(* IEC 61131-3 sources: Mizera_Tube/Plc (part 12) *)

(* ---- mac_func.plc ---- *)
*******************************************************************************
*   MAC_FUNC.PLC
*   ESAutomotion
*   LASER machine
*******************************************************************************
VAR
#include "cnc.inc"
END_VAR

VAR_IN_OUT
#include "mem.inc"
#include "RemContr.inc"
END_VAR

#include "iol.inc"

*******************************************************************************
* function block to manage the override
*******************************************************************************
FUNCTION_BLOCK OVERRIDE

VAR_INPUT
xAnalInput:          DWORD;     * input for potentiometer
xForceLowFeed:       BOOL;      * force the feed to SlowFeed
END_VAR

VAR_OUTPUT
y_Value:             DWORD;
END_VAR

VAR
feedVal:             DWORD;
TON_guiJOG_Min:        TON;   *TON for GUI button JOG to Minus
TON_guiJOG_Max:        TON;   *TON for GUI button JOG to Maximum
TON_BlinkAux_A:	       TON;   *TON Blinking Auxiliar Step A
TON_BlinkAux_B:	       TON;   *TON Blinking Auxiliar Step B
RTRG_guiJOG_Min:    R_TRIG;   *RTRIG for GUI button JOG to Minus
RTRG_guiJOG_Max:    R_TRIG;   *RTRIG for GUI button JOG to Maximum
RTRG_auxBlinkAux:   R_TRIG;
ValOvrr:             DWORD;   *DWORD Calculated value for Override from EncAPos
auxBlinkAux_A:        BOOL;   *BOOL Auxiliar Blinking 150 mseg Step A
auxBlinkAux_B:        BOOL;   *BOOL Auxiliar Blinking 150 mseg Step B
FeedGuiMem:          DWORD;   * support memory for hmi feedrate management
FEED_Minus:           BOOL;
FEED_Plus:            BOOL;

END_VAR
*******************************************************************************

LD   %Type
EQ   0
JMPCN no_analogue_sig

LD   xAnalInput                    ** input for potentiometer
MUL  %MaxPercent
DIV  4095                 *  (16 bit = 32767) [ se 12 bit usare 4095 ]
ST   feedVal              * DWORD Calculated value for Override

JMP  end
no_analogue_sig:

*-----------------------------------------------------------------
* FEED Override by GUI pushbuttons

LD   %Type
EQ   1
JMPCN no_HMI_sig

LD   %PulMinus             ** RTRIG for GUI button JOG to Minus
OR   RemContrFeedMinus     ** Xhc_Puls.13 Feed minus
ST   FEED_Minus

LD   %PulPlus              ** RTRIG for GUI button JOG to Maximum
OR   RemContrFeedPlus      ** Xhc_Puls.9  Feed plus
ST   FEED_Plus

CAL  RTRG_guiJOG_Min(CLK=FEED_Minus) ** RTRIG for GUI button JOG to Minus
CAL  RTRG_guiJOG_Max(CLK=FEED_Plus) ** RTRIG for GUI button JOG to Maximum

CAL  TON_guiJOG_Min(IN=FEED_Minus, PT=%CostK30) ** TON for GUI button JOG to Minus
CAL  TON_guiJOG_Max(IN=FEED_Plus, PT=%CostK30) ** TON for GUI button JOG to Maximum

LDN  TON_BlinkAux_B.Q           ** TON Blinking Auxiliar Step A
ST   auxBlinkAux_A                 ** BOOL Auxiliar Blinking 150 mseg Step A

CAL  TON_BlinkAux_A(IN=auxBlinkAux_A,PT=40) ** TON Blinking Auxiliar Step A
CAL  TON_BlinkAux_B(IN=TON_BlinkAux_A.Q,PT=20) ** TON Blinking Auxiliar Step B

LD   TON_BlinkAux_A.Q           ** TON Blinking Auxiliar Step B
ST   auxBlinkAux_B                 ** BOOL Auxiliar Blinking 150 mseg Step B

CAL  RTRG_auxBlinkAux(CLK=auxBlinkAux_B) ** BOOL Auxiliar Blinking 150 mseg Step B

*
LD   RTRG_guiJOG_Min.Q          ** RTRIG for GUI button JOG to Minus
OR   (
LD   TON_guiJOG_Min.Q           ** TON for GUI button JOG to Minus
AND  RTRG_auxBlinkAux.Q         ** RTRG Auxiliary user asimetric blinking
)
AND  (
LD   FeedGuiMem                    ** support memory for hmi feedrate management
GT   %MinPercent
)
JMPCN No_RTRG_guiJOG_Min
LD   FeedGuiMem                    ** support memory for hmi feedrate management
SUB  %IncStep
ST   FeedGuiMem                    ** support memory for hmi feedrate management
No_RTRG_guiJOG_Min:
*

LD   RTRG_guiJOG_Max.Q          ** RTRIG for GUI button JOG to Maximum
OR   (
LD   TON_guiJOG_Max.Q         ** TON for GUI button JOG to Maximum
AND  RTRG_auxBlinkAux.Q       ** RTRG Auxiliary user asimetric blinking
)
AND  (
LD   FeedGuiMem                    ** support memory for hmi feedrate management
LT   %MaxPercent
)
JMPCN  No_RTRG_guiJOG_Max
LD   FeedGuiMem                    ** support memory for hmi feedrate management
ADD  %IncStep
ST   FeedGuiMem                    ** support memory for hmi feedrate management
No_RTRG_guiJOG_Max:

LD   FeedGuiMem                    ** support memory for hmi feedrate management
ST   feedVal

JMP  end
no_HMI_sig:

end:
*---------------------------------------------------------------------
LD   feedVal
LT   %MinPercent
JMPCN min_feed_limit

LD   %MinPercent
ST   feedVal

min_feed_limit:
LD   xForceLowFeed                 ** force the feed to SlowFeed
JMPCN low_feed
LD   %SlowFeed
ST   feedVal

low_feed:
LD   feedVal
ST   y_Value

END_FUNCTION_BLOCK

*******************************************************************************
* from potentiometer or from HMI
*******************************************************************************
FUNCTION_BLOCK OP_MODE

VAR_INPUT
xSelRef:        BOOL;
xSelSingRef:    BOOL;
xSelJog:        BOOL;
xSelAut:        BOOL;
xSelInc:        BOOL;
xSelMdi:        BOOL;
END_VAR

VAR_OUTPUT
ySelRef:        BOOL;
ySelSingRef:    BOOL;
ySelJog:        BOOL;
ySelAut:        BOOL;
ySelInc:        BOOL;
ySelMdi:        BOOL;
END_VAR

VAR
RTRG_SEL_REF:   R_TRIG;   *Ref state trigger
RTRG_SEL_REF_S: R_TRIG;   *Ref single state trigger
RTRG_SEL_JOG:   R_TRIG;   *Jog state trigger
RTRG_SEL_AUT:   R_TRIG;   *Aut state trigger
RTRG_SEL_INC:   R_TRIG;   *Inc state trigger
RTRG_SEL_MDI:   R_TRIG;   *Mdi state trigger
END_VAR

*******************************************************************************
LD   %rc8.0
JMPC no_change

CAL  RTRG_SEL_REF(CLK=xSelRef)     ** Ref state trigger
CAL  RTRG_SEL_REF_S(CLK=xSelSingRef) ** Ref single state trigger
CAL  RTRG_SEL_JOG(CLK=xSelJog)     ** Jog state trigger
CAL  RTRG_SEL_AUT(CLK=xSelAut)     ** Aut state trigger
CAL  RTRG_SEL_INC(CLK=xSelInc)     ** Inc state trigger
CAL  RTRG_SEL_MDI(CLK=xSelMdi)     ** Mdi state trigger

* Ref
LD   RTRG_SEL_REF.Q
JMPCN no_ref

LD   1
ST   ySelRef

LD   ALWAYS_ONE                    ** PLCFLAGS.1  Flag sempre stato on
ST   PLC_SEL_REF                   ** ui16.1 Selezione Modo REF da Plc

LD   0
ST   ySelJog
ST   ySelAut
ST   ySelInc
ST   ySelMdi
ST   ySelSingRef

no_ref:
LD   RTRG_SEL_REF_S.Q
JMPCN no_refs

LD   1
ST   ySelSingRef

LD   ALWAYS_ONE                    ** PLCFLAGS.1  Flag sempre stato on
ST   PLC_SEL_REF                   ** ui16.1 Selezione Modo REF da Plc

LD   0
ST   ySelJog
ST   ySelAut
ST   ySelInc
ST   ySelMdi

LD   ALWAYS_ONE                    ** PLCFLAGS.1  Flag sempre stato on
ST   PLC_SEL_SINGREF               ** ui16.28 Selezione REF singolo

no_refs:

* Jog
LD   RTRG_SEL_JOG.Q
JMPCN no_jog

LD   1
ST   ySelJog

LD   0
ST   ySelRef
ST   ySelAut
ST   ySelInc
ST   ySelMdi
ST   ySelSingRef

LD   ALWAYS_ZERO                   ** PLCFLAGS.0  Flag sempre stato off
ST   PLC_SEL_REF                   ** ui16.1 Selezione Modo REF da Plc
ST   PLC_SEL_SINGREF               ** ui16.28 Selezione REF singolo

no_jog:
* Auto
LD   RTRG_SEL_AUT.Q
JMPCN no_aut

LD   1
ST   ySelAut

LD   0
ST   ySelRef
ST   ySelInc
ST   ySelJog
ST   ySelMdi
ST   ySelSingRef

LD   ALWAYS_ZERO                   ** PLCFLAGS.0  Flag sempre stato off
ST   PLC_SEL_REF                   ** ui16.1 Selezione Modo REF da Plc
ST   PLC_SEL_SINGREF               ** ui16.28 Selezione REF singolo

no_aut:
* Inc
LD   RTRG_SEL_INC.Q
JMPCN no_Inc

LD   1
ST   ySelInc

LD   0
ST   ySelRef
ST   ySelAut
ST   ySelJog
ST   ySelMdi
ST   ySelSingRef

LD   ALWAYS_ZERO                   ** PLCFLAGS.0  Flag sempre stato off
ST   PLC_SEL_REF                   ** ui16.1 Selezione Modo REF da Plc
ST   PLC_SEL_SINGREF               ** ui16.28 Selezione REF singolo

no_Inc:

* Mdi
LD   RTRG_SEL_MDI.Q
JMPCN no_Mdi

LD   1
ST   ySelMdi

LD   0
ST   ySelRef
ST   ySelAut
ST   ySelJog
ST   ySelInc
ST   ySelSingRef

LD   ALWAYS_ZERO                   ** PLCFLAGS.0  Flag sempre stato off
ST   PLC_SEL_REF                   ** ui16.1 Selezione Modo REF da Plc
ST   PLC_SEL_SINGREF               ** ui16.28 Selezione REF singolo

no_Mdi:
no_change:

END_FUNCTION_BLOCK

*******************************************************************************

VAR
TON_PULRESET_EMERG: TON;            *
TON_START_BTN:      TON;            * Filter
RTRIG_START_BTN:    R_TRIG;         * Trig
TP_START_BTN:       TP;             * Command
RTRIG_STOP_BTN:     R_TRIG;         * Trig
TP_STOP_BTN:        TP;             * Command
RTRIG_RES_BTN:      R_TRIG;         * Trig
TP_RES_BTN:         TP;             * Command
TP_STSERV:          TP;
RTRIG_STSERV:       R_TRIG;
appoggio:           BOOL;           * force the feed to SlowFeed
Jog_X_MENO:         BOOL;           * temp
Jog_X_PIU:          BOOL;           * temp
Jog_Y_MENO:         BOOL;           * temp
Jog_Y_PIU:          BOOL;           * temp
END_VAR

*******************************************************************************
*   Gestione pulsanti e relativi input associati
*******************************************************************************
FUNCTION GEN_BUTTONS

***************************************
* START
***************************************
LD   %ServiceMillePGM.3
OR   %ServiceMillePGM.12
OR   %ServiceMillePGM.13
OR   %ServiceMillePGM.14
OR   ReqCapacitveTest
ST   appoggio
CAL  RTRIG_STSERV(CLK=appoggio)
CAL  TP_STSERV(IN=RTRIG_STSERV.Q,PT=100)

LD   %FUNCBTN.0
OR   I_I_PUL_START                 ** Start
OR   I_I_HW_START                  ** Start (handwheel)
OR   RemContrStart                 ** Xhc_Puls.3  Start push-button
ST   appoggio                      ** force the feed to SlowFeed

CAL  TON_START_BTN(IN=appoggio, PT=100) ** Filter
CAL  RTRIG_START_BTN(CLK=TON_START_BTN.Q) ** Trig
CAL  TP_START_BTN(IN=RTRIG_START_BTN.Q,PT=100) ** Command

LD   TP_START_BTN.Q
OR   TP_STSERV.Q
ST   Pul_Start                     ** (gPlc0.1)Start pushbutton
S    StartButtonPressed
R    HoldButtonPressed

***************************************
* STOP
***************************************
LD   %FUNCBTN.1                    * [Stop]
OR   I_I_PUL_STOP                  ** Stop
OR   I_I_HW_STOP                   ** Stop (handwheel)
OR   RemContrStop                  ** Xhc_Puls.4  Stop push button   *
ST   appoggio                      ** force the feed to SlowFeed

CAL  RTRIG_STOP_BTN(CLK=appoggio)  ** Trig
CAL  TP_STOP_BTN(IN=RTRIG_STOP_BTN.Q,PT=100) ** Command

LD   TP_STOP_BTN.Q
ST   Pul_Stop                      ** (gPlc0.2)Stop pushbutton
S    HoldButtonPressed
R    StartButtonPressed

***************************************
* RESET
***************************************
LD   %FUNCBTN.4
OR   I_I_PUL_RESET                 ** Reset
OR   I_I_HW_RESET                  ** Reset (handwheel)
OR   RemContrReset                 ** Xhc_Puls.5  Reset Push Button
ST   appoggio                      ** force the feed to SlowFeed

CAL  TON_PULRESET_EMERG(IN=appoggio, PT=4000)
LD   TON_PULRESET_EMERG.Q
ST   Pul_Reset_EMERG

CAL  RTRIG_RES_BTN(CLK=appoggio)   ** Trig
LD   RTRIG_RES_BTN.Q
OR   iso_ResetCmd
ST   appoggio

CAL  TP_RES_BTN(IN=appoggio,PT=100) ** Command
LD   TP_RES_BTN.Q
ST   Pul_Reset                     ** (gPlc0.3)Reset pushbutton

LDN  %cn0.rc8.0
ANDN %cn3.rc8.0
JMPCN CLR_RESET
     LD   0
     ST   iso_ResetCmd
CLR_RESET:

***************************************
* [+]
***************************************
LD   %FUNCBTN.2          * [+]
OR(
LD   I_I_HW_JOGPLUS                ** Jog+ (handwheel)
AND  PulsAuxComand                 ** (gPlc2.28)Comando abilitazione da pulsantiera ausiliaria
)
ST   Pul_Jogp                      ** (gPlc0.4)jog+ pushbutton

***************************************
* [-]
***************************************
LD   %FUNCBTN.3          * [-]
OR(
LD   I_I_HW_JOGMINUS               ** jog- (handwheel)
AND  PulsAuxComand                 ** (gPlc2.28)Comando abilitazione da pulsantiera ausiliaria
)
ST   Pul_Jogm                      ** (gPlc0.5)jog- pushbutton

***************************************
*   JOYSTICK MANAGEMENT
*   By keyboard or external inputs
*   %PlcOp0.3 = abilitazione tastiera qwerty
***************************************
LD   %PlcOp0.3                     ** Qwerty keyboard enabled
ST   %ENABFBTN.2           * abilitazioni da PLC Per gestire i tasti movim.Assi(QWERTY)

LD   %PLCFLAGS.0
ST   Jog_X_MENO                    ** temp
ST   Jog_X_PIU                     ** temp
ST   Jog_Y_MENO                    ** temp
ST   Jog_Y_PIU                     ** temp

LD   XxEsaJoy_JOG_Yplus            ** ARRWBTN.1 Pulsanti Jog Joystick
OR   XxEsaJoy_XY_plus              ** ARRWBTN.2 Pulsanti Jog Joystick
OR   XxEsaJoy_XminYpl              ** ARRWBTN.0 Pulsanti Jog Joystick
AND  XxCTRL_ENAB_JOG               ** CTRLBTN.1  CTRL che abilita i pulsanti joystick
JMPCN Next1

LD   UpArrow                       ** (gGui2)Up arrow management
EQ   0
S    Jog_X_MENO                    ** temp

LD   UpArrow                       ** (gGui2)Up arrow management
EQ   1
S    Jog_X_PIU                     ** temp

LD   UpArrow                       ** (gGui2)Up arrow management
EQ   2
S    Jog_Y_MENO                    ** temp

LD   UpArrow                       ** (gGui2)Up arrow management
EQ   3
S    Jog_Y_PIU                     ** temp

Next1:
LD   XxEsaJoy_JOG_Xminus           ** ARRWBTN.3 Pulsanti Jog Joystick
OR   XxEsaJoy_XY_minus             ** ARRWBTN.5 Pulsanti Jog Joystick
OR   XxEsaJoy_XminYpl              ** ARRWBTN.0 Pulsanti Jog Joystick
AND  XxCTRL_ENAB_JOG               ** CTRLBTN.1  CTRL che abilita i pulsanti joystick
JMPCN Next2

LD   LeftArrow                     ** (gGui3)Left arrow management
EQ   0
S    Jog_X_MENO                    ** temp

LD   LeftArrow                     ** (gGui3)Left arrow management
EQ   1
S    Jog_X_PIU                     ** temp

LD   LeftArrow                     ** (gGui3)Left arrow management
EQ   2
S    Jog_Y_MENO                    ** temp

LD   LeftArrow                     ** (gGui3)Left arrow management
EQ   3
S    Jog_Y_PIU                     ** temp

Next2:
LD   XxEsaJoy_JOG_Yminus           ** ARRWBTN.6 Pulsanti Jog Joystick
OR   XxEsaJoy_XY_minus             ** ARRWBTN.5 Pulsanti Jog Joystick
OR   XxEsaJoy_XplYmin              ** ARRWBTN.7 Pulsanti Jog Joystick
AND  XxCTRL_ENAB_JOG               ** CTRLBTN.1  CTRL che abilita i pulsanti joystick
JMPCN Next3

LD   DownArrow                     ** (gGui4)Down arrow management
EQ   0
S    Jog_X_MENO                    ** temp

LD   DownArrow                     ** (gGui4)Down arrow management
EQ   1
S    Jog_X_PIU                     ** temp

LD   DownArrow                     ** (gGui4)Down arrow management
EQ   2
S    Jog_Y_MENO                    ** temp

LD   DownArrow                     ** (gGui4)Down arrow management
EQ   3
S    Jog_Y_PIU                     ** temp

Next3:
LD   XxEsaJoy_JOG_Xplus            ** ARRWBTN.4 Pulsanti Jog Joystick
OR   XxEsaJoy_XY_plus              ** ARRWBTN.2 Pulsanti Jog Joystick
OR   XxEsaJoy_XplYmin              ** ARRWBTN.7 Pulsanti Jog Joystick
AND  XxCTRL_ENAB_JOG               ** CTRLBTN.1  CTRL che abilita i pulsanti joystick
JMPCN Next4

LD   RightArrow                    ** (gGui5)Right arrow management
EQ   0
S    Jog_X_MENO                    ** temp

LD   RightArrow                    ** (gGui5)Right arrow management
EQ   1
S    Jog_X_PIU                     ** temp

LD   RightArrow                    ** (gGui5)Right arrow management
EQ   2
S    Jog_Y_MENO                    ** temp

LD   RightArrow                    ** (gGui5)Right arrow management
EQ   3
S    Jog_Y_PIU                     ** temp

Next4:
LD   Jog_X_PIU                     ** temp
OR   I_I_JOY_X_P                   ** X+ (Joystick)
OR   RemContrXPlus                 ** Xhc_Puls.24 Jog X axis plus         *
ST   JOY_X_P                       ** (gPlc0.14)Joystik X + selezionato

LD   Jog_Y_PIU                     ** temp
OR   I_I_JOY_Y_P                   ** Y+ (Joystick)
OR   RemContrYPlus                 ** Xhc_Puls.22 Jog Y axis plus
ST   JOY_Y_P                       ** (gPlc0.16)Joystik Y + selezionato

LD   Jog_X_MENO                    ** temp
OR   I_I_JOY_X_M                   ** X- (Joystick)
OR   RemContrXMinus                ** Xhc_Puls.22 Jog X axis minus        *
ST   JOY_X_M                       ** (gPlc0.15)Joystik X - selezionato

LD   Jog_Y_MENO                    ** temp
OR   I_I_JOY_Y_M                   ** Y- (Joystick)
OR   RemContrYMinus                ** Xhc_Puls.24 Jog Y axis minus
ST   JOY_Y_M                       ** (gPlc0.17)Joystik Y - selezionato

LD   RemContrUMinus                ** Xhc_Puls.19 Jog U axis minus
ANDN Rem_Combination
OR   Gui_Pul_X_M
ST   JOY_U_M					   **(gPlc2.8)Joystik U - selezionato

LD   RemContrUPlus                 ** Xhc_Puls.27 Jog U axis plus
ANDN Rem_Combination
OR   Gui_Pul_X_P
ST   JOY_U_P                       **(gPlc2.7)Joystik U + selezionato

LD   RemContrCMinus                ** Xhc_Puls.18 Jog C axis minus
ANDN Rem_Combination
ANDN RemContrStop
ST   JOY_C_M                       **(gPlc2.10)Joystik C - selezionato
LD   RemContrCPlus                 ** Xhc_Puls.26 Jog C axis plus
ANDN Rem_Combination
ANDN RemContrStop
ST   JOY_C_P					   **(gPlc2.9)Joystik C + selezionato

LD   RemContrZMinus                ** Xhc_Puls.28 Jog Z axis minus
ANDN Rem_Combination
ST   JOY_Z_M                       **(gPlc19.4)Joystik Z - selezionato

LD   RemContrZPlus                 ** Xhc_Puls.20 Jog Z axis plus
ANDN Rem_Combination
ST   JOY_Z_P					   **(gPlc19.3)Joystik Z + selezionato

END_FUNCTION

(* ---- Mand.plc ---- *)
* Blocchi gestione mandrini da PLC

#funcdec "assi.plc"

VAR
#include "assi.inc"
#include "cnc.inc"
END_VAR

* ----------------------------------------------------------------*
* Blocco Funzionale conversione da numero utensile a numero pocket
* ----------------------------------------------------------------*

FUNCTION_BLOCK SP_TOOL_POCKET

VAR_INPUT
xax_TOOL:     BYTE; * Numero utensile
END_VAR

VAR_OUTPUT
yax_POCKET:   BYTE; * Numero pocket
END_VAR

VAR
INDEX: DWORD;    * Indice per caricamento pocket associato al tool richiesto
END_VAR

* Seleziona il revolver richiesto
PATH %mag[CC_RV]                   ** cc26 Numero magazzino utensile associato al canale

* Se il target è nullo, lo trasferisce allo slave che darà errore
LD   xax_TOOL                      ** Numero utensile
EQ   0
JMPC DIRECT_TOOL

LD   xax_TOOL                      ** Numero utensile
SUB  1
ST   INDEX                         ** Indice per caricamento pocket associato al tool richiesto

* Seleziona il pocket relativo all'utensile richiesto
LD   %tp.map[INDEX]                ** Indice per caricamento pocket associato al tool richiesto
ST   INDEX                         ** Indice per caricamento pocket associato al tool richiesto

* Se il pocket è nullo, usa il numero dell'utensile
LD   INDEX                         ** Indice per caricamento pocket associato al tool richiesto
EQ   0
JMPC DIRECT_TOOL

LD   INDEX                         ** Indice per caricamento pocket associato al tool richiesto
ST   yax_POCKET                    ** Numero pocket

JMP  END_TOOL

DIRECT_TOOL:

LD   xax_TOOL                      ** Numero utensile
ST   yax_POCKET                    ** Numero pocket

END_TOOL:

END_FUNCTION_BLOCK

* ----------------------------------------------------------------*
* Blocco Funzionale conversione da numero pocket a numero utensile
* ----------------------------------------------------------------*

FUNCTION_BLOCK SP_POCKET_TOOL

VAR_INPUT
xax_POCKET:   BYTE; * Numero pocket
END_VAR

VAR_OUTPUT
yax_TOOL:     BYTE; * Numero utensile
END_VAR

VAR
INDEX: DWORD;    * Indice per caricamento tool associato al pocket richiesto
END_VAR

* Seleziona il revolver richiesto
PATH %mag[CC_RV]                   ** cc26 Numero magazzino utensile associato al canale

* Trova l'utensile corrispondente al pocket corrente
LD   0
ST   INDEX                         ** Indice per caricamento tool associato al pocket richiesto

LOOP_POCKET:

LD   %tp.map[INDEX]                ** Indice per caricamento tool associato al pocket richiesto
EQ   xax_POCKET                    ** Numero pocket
JMPC END_POCKET

LD   INDEX                         ** Indice per caricamento tool associato al pocket richiesto
ADD  1
ST   INDEX                         ** Indice per caricamento tool associato al pocket richiesto

LD   INDEX                         ** Indice per caricamento tool associato al pocket richiesto
LT   6
JMPC LOOP_POCKET

* Se l'utensile non è configurato, ritorna utensile pari a zero
LD   -1
ST   INDEX                         ** Indice per caricamento tool associato al pocket richiesto

END_POCKET:

LD   INDEX                         ** Indice per caricamento tool associato al pocket richiesto
ADD  1
ST   yax_TOOL                      ** Numero utensile

END_FUNCTION_BLOCK

* --------------------------------------------*
* Blocco Funzionale posizionamento mandrino
* --------------------------------------------*

FUNCTION_BLOCK SP_POSIZ

VAR_INPUT
xax_ENABLE:   BOOL;       * abilita FB
xax_START:    BOOL;       * start richiesta azione
xax_CLEAR:    BOOL;       * conferma fine comando
xax_IMMDATA:  BOOL;       * dati (quota, vel, toll) immediati
                          * 0 = carica dati di sistema
                          * 1 = carica dati da input FB
xax_INCMODE:  BOOL;       * 0 = assoluto, 1 = incrementale
xax_REVMODE:  BOOL;       * 0 = M19, 1 = orienta per innesto revolver
xax_TOOL:     DWORD;      * Utensile corrente 1-12
xax_QUOTA:    DWORD;      * Quota target assoluta ( 0.1 deg )
xax_VEL:      DWORD;      * Velocita' posizionamento ( rpm )
xax_VSTOP:    DWORD;      * Velocita' di arresto ( rpm )
xax_TOLLP:    DWORD;      * Tolleranza ( 0.1 deg )

END_VAR

VAR_OUTPUT
yax_READY:    BOOL;       * FB pronto per START
yax_RUNNING:  BOOL;       * Esecuzione FB in corso
yax_ENDOK:    BOOL;       * Comando terminato correttamente
yax_ENDERR:   BOOL;       * Comando terminato non correttamente
yax_ERRCODE:  DWORD;      * codice errore ( maschera bit )
END_VAR

VAR
AXFB: AX_COMMAND;
PTFB: SP_POCKET_TOOL;
INDEX: DWORD;    * Indice per caricamento dinamica associata al tool richiesto
END_VAR

* Chiamata FB standard gestione comandi slave

LD   xax_ENABLE                    ** abilita FB
ST   AXFB.xax_ENABLE

LD   xax_START                     ** start richiesta azione
ST   AXFB.xax_START

LD   xax_CLEAR                     ** conferma fine comando
ST   AXFB.xax_CLEAR

CAL  AXFB

* Comando uscite da FB standard

LD   AXFB.yax_READY
ST   yax_READY                     ** FB pronto per START

LD   AXFB.yax_RUNNING
ST   yax_RUNNING                   ** Esecuzione FB in corso

LD   AXFB.yax_ENDOK
ST   yax_ENDOK                     ** Comando terminato correttamente

LD   AXFB.yax_ENDERR
ST   yax_ENDERR                    ** Comando terminato non correttamente

LD   AXFB.yax_ERRCODE
ST   yax_ERRCODE                   ** codice errore ( maschera bit )

*** TRASFERIMENTO DEI REGISTRI FB ALLO SLAVE ***

LD   AXFB.yax_TRDATA
JMPCN END_DATA

LD   xax_INCMODE                   ** 0 = assoluto, 1 = incrementale
JMPC INCMODE

LD   4
ST   FB_CODE                       ** fb0 Codice Operativo comando

JMP  END_INCMODE

INCMODE:

LD   5
ST   FB_CODE                       ** fb0 Codice Operativo comando

END_INCMODE:

LD   xax_IMMDATA                   ** dati (quota, vel, toll) immediati
JMPC IMMDATA

LD   xax_REVMODE                   ** 0 = M19, 1 = orienta per innesto revolver
JMPC REVMODE

LD   CO_ANGM19                     ** rc38 Angolo orientamento mandrino M19
ST   FB_QUOTADEG                   ** fb1 Quota target assoluta (0.1 deg)

JMP  END_REVMODE

REVMODE:

* Seleziona il revolver richiesto
PATH %mag[CC_RV]                   ** cc26 Numero magazzino utensile associato al canale

LD   RV_PARKQTA                    ** prv11 Quota di parcheggio
ST   FB_QUOTADEG                   ** fb1 Quota target assoluta (0.1 deg)

END_REVMODE:

* Se non è configurato il revolver, usa i dati del mandrino
LD   CC_MAG                        ** cc25 Tipo magazzino utensile (1=revolver)
NE   1
JMPC MAND_DATA

* Trova l'utensile corrispondente al pocket corrente
CAL  PTFB(xax_POCKET=xax_TOOL)     ** Utensile corrente 1-12

* Se l'utensile non è configurato, usa i dati di default del mandrino
LD   PTFB.yax_TOOL
EQ   0
JMPC MAND_DATA

LD   PTFB.yax_TOOL
SUB  1
ST   INDEX                         ** Indice per caricamento dinamica associata al tool richiesto

* Seleziona i dati mandrino relativi all'utensile corrente
LD   %tp.dyn[INDEX]                ** Indice per caricamento dinamica associata al tool richiesto
ST   INDEX                         ** Indice per caricamento dinamica associata al tool richiesto

PATH %tdyn[INDEX]                  ** Indice per caricamento dinamica associata al tool richiesto

LD   TDYN_VELPOS                   ** dy7 Velocità in orientamento (rpm)
ST   FB_VELRPM                     ** fb2 Velocita' posizionamento (rpm)

LD   TDYN_VELPOS                   ** dy7 Velocità in orientamento (rpm)
ST   FB_VSTOP                      ** fb3 Velocita' arresto mandrino (rpm)

LD   TDYN_TOLLERF                  ** dy6 Quota di tolleranza fine (gradi)
ST   FB_TOLLDEG                    ** fb7 Tolleranza (0.1 deg)

JMP  END_DATA

MAND_DATA:

LD   SP_VELM19                     ** pa37 Velocità mandrino in orientamento (rpm)
ST   FB_VELRPM                     ** fb2 Velocita' posizionamento (rpm)

LD   SP_VELM19                     ** pa37 Velocità mandrino in orientamento (rpm)
ST   FB_VSTOP                      ** fb3 Velocita' arresto mandrino (rpm)

LD   SP_TOLLERG                    ** pa6 Quota tolleranza grossolana
ST   FB_TOLLDEG                    ** fb7 Tolleranza (0.1 deg)

JMP  END_DATA

IMMDATA:

LD   xax_QUOTA                     ** Quota target assoluta ( 0.1 deg )
ST   FB_QUOTADEG                   ** fb1 Quota target assoluta (0.1 deg)

LD   xax_VEL                       ** Velocita' posizionamento ( rpm )
ST   FB_VELRPM                     ** fb2 Velocita' posizionamento (rpm)

LD   xax_VSTOP                     ** Velocita' di arresto ( rpm )
ST   FB_VSTOP                      ** fb3 Velocita' arresto mandrino (rpm)

LD   xax_TOLLP                     ** Tolleranza ( 0.1 deg )
ST   FB_TOLLDEG                    ** fb7 Tolleranza (0.1 deg)

END_DATA:

END_FUNCTION_BLOCK

* ----------------------------------------------*
* Blocco Funzionale qualifica mandrino/ revolver
* ----------------------------------------------*

FUNCTION_BLOCK SP_QUALIFY

VAR_INPUT
xax_ENABLE:   BOOL;       * abilita FB
xax_START:    BOOL;       * start richiesta azione
xax_CLEAR:    BOOL;       * conferma fine comando
xax_IMMDATA:  BOOL;       * dati (vel, rampe, gain) immediati
                          * 0 = carica dati di sistema
                          * 1 = carica dati da input FB
xax_REVMODE:  BOOL;       * 0 = qualifica mandrino, 1 = qualifica revolver
xax_PRESET:   BOOL;       * Abilita preset automatico mandrino
xax_TOOL:     DWORD;      * Utensile corrente 1-12
xax_VMAX:     DWORD;      * Velocita' massima ( rpm )
xax_ACCEL:    DWORD;      * Accelerazione (msec o rev/s2)
xax_DECEL:    DWORD;      * Decelerazione (msec o rev/s2)
xax_RAMPES:   DWORD;      * Tempo Rampe S (msec o rev/s3)
xax_GAINP:    DWORD;      * Guadagno P (0.001 DAC/pulses o 0.001 sec-1)
xax_FLWER:    DWORD;      * Errore inseguimento massimo (pulses o 0.001 rev)
xax_EFS:      DWORD;      * Tensione di fondo scala (mV)

END_VAR

VAR_OUTPUT
yax_READY:    BOOL;       * FB pronto per START
yax_RUNNING:  BOOL;       * Esecuzione FB in corso
yax_ENDOK:    BOOL;       * Comando terminato correttamente
yax_ENDERR:   BOOL;       * Comando terminato non correttamente
yax_ERRCODE:  DWORD;      * codice errore ( maschera bit )
END_VAR

VAR
AXFB: AX_COMMAND;
PTFB: SP_POCKET_TOOL;
INDEX: DWORD;    * Indice per caricamento dinamica associata al tool richiesto
END_VAR

* Chiamata FB standard gestione comandi slave

LD   xax_ENABLE                    ** abilita FB
ST   AXFB.xax_ENABLE

LD   xax_START                     ** start richiesta azione
ST   AXFB.xax_START

LD   xax_CLEAR                     ** conferma fine comando
ST   AXFB.xax_CLEAR

CAL  AXFB

* Comando uscite da FB standard

LD   AXFB.yax_READY
ST   yax_READY                     ** FB pronto per START

LD   AXFB.yax_RUNNING
ST   yax_RUNNING                   ** Esecuzione FB in corso

LD   AXFB.yax_ENDOK
ST   yax_ENDOK                     ** Comando terminato correttamente

LD   AXFB.yax_ENDERR
ST   yax_ENDERR                    ** Comando terminato non correttamente

LD   AXFB.yax_ERRCODE
ST   yax_ERRCODE                   ** codice errore ( maschera bit )

*** TRASFERIMENTO DEI REGISTRI FB ALLO SLAVE ***

LD   AXFB.yax_TRDATA
JMPCN END_DATA

LD   xax_REVMODE                   ** 0 = qualifica mandrino, 1 = qualifica revolver
JMPC REVMODE

LD   xax_PRESET                    ** Abilita preset automatico mandrino
JMPC MANPRESET

LD   3
ST   FB_CODE                       ** fb0 Codice Operativo comando

JMP  END_REVMODE

MANPRESET:

LD   20
ST   FB_CODE                       ** fb0 Codice Operativo comando

JMP  END_REVMODE

REVMODE:

LD   xax_PRESET                    ** Abilita preset automatico mandrino
JMPC REVPRESET

LD   6
ST   FB_CODE                       ** fb0 Codice Operativo comando

JMP  END_REVMODE

REVPRESET:

LD   21
ST   FB_CODE                       ** fb0 Codice Operativo comando

END_REVMODE:

LD   xax_TOOL                      ** Utensile corrente 1-12
ST   FB_TOOL                       ** fb1 Numero utensile corrente 1-12

LD   xax_IMMDATA                   ** dati (vel, rampe, gain) immediati
JMPC IMMDATA

LD   xax_REVMODE                   ** 0 = qualifica mandrino, 1 = qualifica revolver
JMPC REVPAR

* Trova l'utensile corrispondente al pocket corrente
CAL  PTFB(xax_POCKET=xax_TOOL)     ** Utensile corrente 1-12

* Se l'utensile non è configurato, usa i dati di default del mandrino
LD   PTFB.yax_TOOL
EQ   0
JMPC MAND_DATA

LD   PTFB.yax_TOOL
SUB  1
ST   INDEX                         ** Indice per caricamento dinamica associata al tool richiesto

* Seleziona i dati mandrino relativi all'utensile corrente
LD   %tp.dyn[INDEX]                ** Indice per caricamento dinamica associata al tool richiesto
ST   INDEX                         ** Indice per caricamento dinamica associata al tool richiesto

PATH %tdyn[INDEX]                  ** Indice per caricamento dinamica associata al tool richiesto

LD   TDYN_VELLIM                   ** dy0 Velocità limite
ST   FB_VMAXRPM                    ** fb3 Velocita' massima (rpm)

LD   TDYN_ACCTIME                  ** dy1 Tempo accelerazione
ST   FB_ACCELREV                   ** fb4 Accelerazione (msec o rev/s2)

LD   TDYN_DECTIME                  ** dy2 Tempo decelerazione
ST   FB_DECELREV                   ** fb5 Decelerazione (msec o rev/s2)

LD   TDYN_DELAYS                   ** dy3 Tempo di rampa S
ST   FB_RAMPESREV                  ** fb6 Tempo Rampe S (msec o rev/s3)

LD   TDYN_GAINP                    ** dy4 Guadagno P
ST   FB_GAINP                      ** fb8 Guadagno P (0.001 DAC/pulses o 0.001 sec-1)

LD   TDYN_FWERR                    ** dy5 Massimo errore inseguimento
ST   FB_FLWERREV                   ** fb9 Errore inseguimento limite (pulses o 0.001 rev)

LD   DC_DACREF                     ** dDacRef Tensione a Vel. Max (mVolt)
ST   FB_EFS                        ** fb11 Tensione di fondo scala (mV)

JMP  END_DATA

MAND_DATA:

LD   SP_VELMAX                     ** pa9 Velocità massima
ST   FB_VMAXRPM                    ** fb3 Velocita' massima (rpm)

LD   SP_ACCEL                      ** pa1 Accelerazione massima
ST   FB_ACCELREV                   ** fb4 Accelerazione (msec o rev/s2)

LD   SP_DECEL                      ** pa2 Decelerazione massima
ST   FB_DECELREV                   ** fb5 Decelerazione (msec o rev/s2)

LD   SP_JERK                       ** pa25 Jerk massimo
ST   FB_RAMPESREV                  ** fb6 Tempo Rampe S (msec o rev/s3)

LD   SP_KPGAIN                     ** pa10 Guadagno P
ST   FB_GAINP                      ** fb8 Guadagno P (0.001 DAC/pulses o 0.001 sec-1)

LD   SP_SSERR                      ** pa5 Errore inseguimento massimo
ST   FB_FLWERREV                   ** fb9 Errore inseguimento limite (pulses o 0.001 rev)

LD   DC_DACREF                     ** dDacRef Tensione a Vel. Max (mVolt)
ST   FB_EFS                        ** fb11 Tensione di fondo scala (mV)

JMP  END_DATA

REVPAR:

PATH %mag[CC_RV]                   ** cc26 Numero magazzino utensile associato al canale

LD   RV_VELLIM                     ** prv3 Velocità limite revolver (rpm)
ST   FB_VMAXRPM                    ** fb3 Velocita' massima (rpm)

LD   RV_ACCTIME                    ** prv4 Tempo accelerazione
ST   FB_ACCELREV                   ** fb4 Accelerazione (msec o rev/s2)

LD   RV_DECTIME                    ** prv5 Tempo decelerazione
ST   FB_DECELREV                   ** fb5 Decelerazione (msec o rev/s2)

LD   RV_DELAYS                     ** prv6 Tempo di rampa S
ST   FB_RAMPESREV                  ** fb6 Tempo Rampe S (msec o rev/s3)

LD   RV_GAINP                      ** prv7 Guadagno P
ST   FB_GAINP                      ** fb8 Guadagno P (0.001 DAC/pulses o 0.001 sec-1)

LD   RV_FWERR                      ** prv8 Massimo errore inseguimento
ST   FB_FLWERREV                   ** fb9 Errore inseguimento limite (pulses o 0.001 rev)

LD   DC_DACREF                     ** dDacRef Tensione a Vel. Max (mVolt)
ST   FB_EFS                        ** fb11 Tensione di fondo scala (mV)

JMP  END_DATA

IMMDATA:

LD   xax_VMAX                      ** Velocita' massima ( rpm )
ST   FB_VMAXRPM                    ** fb3 Velocita' massima (rpm)

LD   xax_ACCEL                     ** Accelerazione (msec o rev/s2)
ST   FB_ACCELREV                   ** fb4 Accelerazione (msec o rev/s2)

LD   xax_DECEL                     ** Decelerazione (msec o rev/s2)
ST   FB_DECELREV                   ** fb5 Decelerazione (msec o rev/s2)

LD   xax_RAMPES                    ** Tempo Rampe S (msec o rev/s3)
ST   FB_RAMPESREV                  ** fb6 Tempo Rampe S (msec o rev/s3)

LD   xax_GAINP                     ** Guadagno P (0.001 DAC/pulses o 0.001 sec-1)
ST   FB_GAINP                      ** fb8 Guadagno P (0.001 DAC/pulses o 0.001 sec-1)

LD   xax_FLWER                     ** Errore inseguimento massimo (pulses o 0.001 rev)
ST   FB_FLWERREV                   ** fb9 Errore inseguimento limite (pulses o 0.001 rev)

LD   xax_EFS                       ** Tensione di fondo scala (mV)
ST   FB_EFS                        ** fb11 Tensione di fondo scala (mV)

END_DATA:

END_FUNCTION_BLOCK

* --------------------------------------------*
* Blocco Funzionale posizionamento revolver
* --------------------------------------------*

FUNCTION_BLOCK SP_POSREV

VAR_INPUT
xax_ENABLE:   BOOL;       * abilita FB
xax_START:    BOOL;       * start richiesta azione
xax_CLEAR:    BOOL;       * conferma fine comando
xax_IMMDATA:  BOOL;       * dati (vmax, toll) immediati
                          * 0 = carica dati di sistema
                          * 1 = carica dati da input FB
xax_INCFORW:  BOOL;       * 0 = assoluto, 1 = incrementale avanti
xax_INCBACK:  BOOL;       * 0 = assoluto, 1 = incrementale indietro
xax_TARGR:    DWORD;      * Posizione target (1-12)
xax_SLOW:     BOOL;       * 0 = veloce, 1 = lento
xax_VEL:      DWORD;      * Velocita' posizionamento ( rpm )
xax_TOLLP:    DWORD;      * Tolleranza ( 0.1 deg )

END_VAR

VAR_OUTPUT
yax_READY:    BOOL;       * FB pronto per START
yax_RUNNING:  BOOL;       * Esecuzione FB in corso
yax_ENDOK:    BOOL;       * Comando terminato correttamente
yax_ENDERR:   BOOL;       * Comando terminato non correttamente
yax_ERRCODE:  DWORD;      * codice errore ( maschera bit )
END_VAR

VAR
AXFB: AX_COMMAND;
TPFB: SP_TOOL_POCKET;
END_VAR

* Chiamata FB standard gestione comandi slave

LD   xax_ENABLE                    ** abilita FB
ST   AXFB.xax_ENABLE

LD   xax_START                     ** start richiesta azione
ST   AXFB.xax_START

LD   xax_CLEAR                     ** conferma fine comando
ST   AXFB.xax_CLEAR

CAL  AXFB

* Comando uscite da FB standard

LD   AXFB.yax_READY
ST   yax_READY                     ** FB pronto per START

LD   AXFB.yax_RUNNING
ST   yax_RUNNING                   ** Esecuzione FB in corso

LD   AXFB.yax_ENDOK
ST   yax_ENDOK                     ** Comando terminato correttamente

LD   AXFB.yax_ENDERR
ST   yax_ENDERR                    ** Comando terminato non correttamente

LD   AXFB.yax_ERRCODE
ST   yax_ERRCODE                   ** codice errore ( maschera bit )

*** TRASFERIMENTO DEI REGISTRI FB ALLO SLAVE ***

LD   AXFB.yax_TRDATA
JMPCN END_DATA

LD   xax_INCFORW                   ** 0 = assoluto, 1 = incrementale avanti
OR   xax_INCBACK                   ** 0 = assoluto, 1 = incrementale indietro
JMPC INCMODE

LD   7
ST   FB_CODE                       ** fb0 Codice Operativo comando

* Trova il pocket corrispondente all'utensile target
CAL  TPFB(xax_TOOL=xax_TARGR)      ** Posizione target (1-12)

LD   TPFB.yax_POCKET
ST   FB_TARGR                      ** fb10 Numero utensile target (1-12)

JMP  END_INCMODE

INCMODE:

* Seleziona il revolver richiesto
PATH %mag[CC_RV]                   ** cc26 Numero magazzino utensile associato al canale

LD   8
ST   FB_CODE                       ** fb0 Codice Operativo comando

LD   xax_INCFORW                   ** 0 = assoluto, 1 = incrementale avanti
JMPCN INCMENO

LD   1
ST   FB_TARGR                      ** fb10 Numero utensile target (1-12)

JMP  END_INCMODE

INCMENO:

LD   -1
ST   FB_TARGR                      ** fb10 Numero utensile target (1-12)

END_INCMODE:

LD   xax_IMMDATA                   ** dati (vmax, toll) immediati
JMPC IMMDATA

LD   xax_SLOW                      ** 0 = veloce, 1 = lento
JMPC SINGCYC

LD   RV_VELPOS                     ** prv12 Velocità in orientamento
ST   FB_VELRPM                     ** fb2 Velocita' posizionamento (rpm)

JMP  END_SINGCYC

SINGCYC:

LD   RV_VELCYCLE                   ** prv14 Velocità in SINGLE CYCLE
ST   FB_VELRPM                     ** fb2 Velocita' posizionamento (rpm)

END_SINGCYC:

LD   RV_TOLLERF                    ** prv9 Quota di tolleranza fine (gradi)
ST   FB_TOLLDEG                    ** fb7 Tolleranza (0.1 deg)

JMP  END_DATA

IMMDATA:

LD   xax_VEL                       ** Velocita' posizionamento ( rpm )
ST   FB_VELRPM                     ** fb2 Velocita' posizionamento (rpm)

LD   xax_TOLLP                     ** Tolleranza ( 0.1 deg )
ST   FB_TOLLDEG                    ** fb7 Tolleranza (0.1 deg)

END_DATA:

END_FUNCTION_BLOCK

* ----------------------------------------------*
* Funzione selezione velocità rotazione mandrino
* ----------------------------------------------*

FUNCTION SP_SELSPEED

LD   BCI_JOGOPEN                   ** rc0.22  Abilita esecuzione JOG a Loop Aperto
AND  BCI_MAN                       ** rc0.9  Selettore modi operativi su JOG (manuale)
ST   BAI_VOLTS                     ** ra0.31 Rotaz. speed in Volts (JOG open mandrino)

LD   BCI_MDI                       ** rc0.11  Selettore modi operativi su MDI (semiautom)
OR   BCI_AUT                       ** rc0.12  Selettore modi operativi su AUT (automatic)
JMPC VELAUT

LD   BAO_REVOL                     ** ra3.31 Selezione mandrino come revolver
JMPC VELJOGREVO

LD   BCI_TAR                       ** rc0.8  Selettore modi operativi su REF (taratura)
JMPC VELREFMAND

LD   BAI_VOLTS                     ** ra0.31 Rotaz. speed in Volts (JOG open mandrino)
JMPC VELJOGOPEN

LD   SP_VELJOG                     ** pa36 Velocità JOG mandrino (rpm)
ST   AI_SPEED                      ** ra32 Velocità rotazione al mandrino (rpm)

JMP END_VELMAND

VELJOGOPEN:

LD   CI_JOGOPEN                    ** rc5  Tensione JOG a Loop Aperto
ST   AI_SPEED                      ** ra32 Velocità rotazione al mandrino (rpm)

JMP END_VELMAND

VELREFMAND:

LD   BAI_FCRALL                    ** ra0.13 Finecorsa Taratura
JMPC RICTACCAMAND

LD   SP_VELMICRO                   ** pa19 Velocità ricerca micro mandrino (rpm)
ST   AI_SPEED                      ** ra32 Velocità rotazione al mandrino (rpm)

JMP END_VELMAND

RICTACCAMAND:

LD   SP_VELTACCA                   ** pa20 Velocità ricerca tacca mandrino (rpm)
ST   AI_SPEED                      ** ra32 Velocità rotazione al mandrino (rpm)

JMP END_VELMAND

VELJOGREVO:

* Seleziona il revolver richiesto
PATH %mag[CC_RV]                   ** cc26 Numero magazzino utensile associato al canale

LD   RV_VELJOG                     ** prv13 Velocità in JOG
ST   AI_SPEED                      ** ra32 Velocità rotazione al mandrino (rpm)

JMP END_VELMAND

VELAUT:

LD   CUR_SPIN3                     ** rg0.4 Mandrino corrente = S3
JMPCN MAND2

LD   CO_VELMANDS3                  ** rc82 Velocità mandrino 3 richiesta da canale (funzione S)
ST   AI_SPEED                      ** ra32 Velocità rotazione al mandrino (rpm)

JMP  END_VELMAND

MAND2:

LD   CUR_SPIN2                     ** rg0.3 Mandrino corrente = S2
JMPCN MAND1

LD   CO_VELMANDS2                  ** rc81 Velocità mandrino 2 richiesta da canale (funzione S)
ST   AI_SPEED                      ** ra32 Velocità rotazione al mandrino (rpm)

JMP  END_VELMAND

MAND1:

LD   CO_VELMAND                    ** rc25 Velocità mandrino 1 richiesta da canale (funzione S)
ST   AI_SPEED                      ** ra32 Velocità rotazione al mandrino (rpm)

END_VELMAND:

END_FUNCTION
